// TIA Portal V20 export
DATA_BLOCK "GLOBAL_SERVICE_DB"   // DB218
{ S7_Optimized_Access := 'TRUE' }
// stored: AutoNumber false, MemoryReserve 100
   VAR RETAIN
      Service_Req : Array[0..10] of "ROBOT_GLOBAL_SRV_UDT";
   END_VAR
BEGIN
   // Service_Req[5] : OPMODE5
   // Service_Req[6] : OPMODE6
END_DATA_BLOCK
